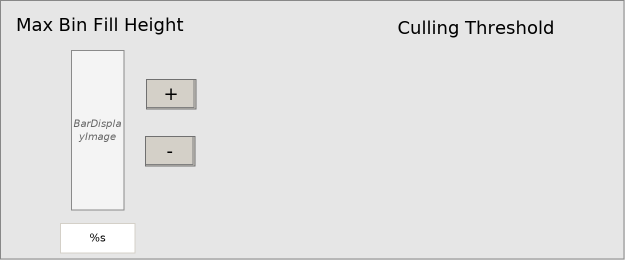
VISUALIZATION BinFiller  // 625x260
    Textfield (0,10 200x30), "Max Bin Fill Height"
    Textfield (60,223 75x30), "%s"
    BarDisplayImage (71,50 53x160), style: BarDisplayImage-Gray, scale format: %.0f, scale 0..100
    Button (146,79 50x30), "+"
    Button (145,136 50x30), "-"
    Textfield (376,13 200x30), "Culling Threshold"
END_VISUALIZATION

(* stored: Version 1.1.0.1, ProductVersion 3.1.4024.15
   Visu BinFiller: Id {09bbd1c1-6caa-40b9-b718-c7d340983037} *)
